// TwinCAT 3 PLC project Untitled1
// ProgramVersion: 3.1.4023.0
// libraries:
//   CmpBitmapPool, * (System)
//   Tc2_MC2, * (Beckhoff Automation GmbH)
//   Tc2_Standard, * (Beckhoff Automation GmbH)
//   Tc2_System, * (Beckhoff Automation GmbH)
//   Tc2_Utilities, * (Beckhoff Automation GmbH)
//   Tc3_Module, * (Beckhoff Automation GmbH)
// project tree:
//   DUTs/ A21ToolStorage.TcDUT (not stored), Bundle.TcDUT (not stored), EOAT.TcDUT (not stored), Interval.TcDUT (not stored), PositionMaterials.TcDUT (not stored)
//   DUTs/Enums/ A21.TcDUT (not stored), Chipboard.TcDUT (not stored), Homing.TcDUT, SectionEnum.TcDUT (not stored), Surface.TcDUT (not stored), WoodBunk.TcDUT (not stored)
//   DUTs/Insertion/Drives/ AirPiston.TcPOU (not stored), ClearLinkMC.TcPOU, SimplePiston.TcPOU (not stored)
//   DUTs/Insertion/ Insertion.TcPOU (not stored), SuctionPad.TcDUT (not stored)
//   DUTs/Insertion/Prototypes/ FBA_Drive.TcPOU (not stored), I_ContinuousDrive.TcIO (not stored), I_Drive.TcIO (not stored), I_PositionalDrive.TcIO (not stored), I_EncodedDrive.TcIO (not stored)
//   DUTs/Machines/ Conveyor.TcPOU (not stored), ConveyorMode.TcDUT (not stored), KukaRobot.TcPOU (not stored), RobotA21.TcPOU (not stored), StrapMachine.TcPOU
//   DUTs/Material Holders/ MaterialHolder.TcPOU, MaterialSlot.TcDUT, SkidMagazine.TcPOU, StagingTable.TcPOU
//   GVLs/ ContainerArrays.TcGVL, GVL.TcGVL (not stored), Hardware.TcGVL (not stored), Misc.TcGVL (not stored)
//   / PlcTask.TcTTO (not stored)
//   POUs/A21a - Chipboard/AOIs/ AOI_LoadChipboard.TcPOU
//   POUs/A21b - Wood Bunk/AOIs/ AOI_LoadWoodBunk.TcPOU, AOI_StageWoodBunk.TcPOU, AOI_StagingTemplate.TcPOU
//   POUs/ FB_System.TcPOU (not stored), MAIN.TcPOU
//   POUs/Hardware Calls/ InsertionQuality.TcPOU (not stored), SuctionQuality.TcPOU (not stored), CallHardware.TcPOU, SetSuctions.TcPOU (not stored), SetupHardware.TcPOU
//   POUs/A21a - Chipboard/ ChipboardEx.TcPOU
//   POUs/A21b - Wood Bunk/ WoodBunkEx.TcPOU
//   POUs/Utility/ AddToStringArray.TcPOU (not stored), ArrayIsEmpty.TcPOU (not stored), BoolVLArrayToInteger.TcPOU (not stored), BoolPtrArrayToInteger.TcPOU (not stored), CleanStringsArray.TcPOU (not stored), IntegerBitAccess.TcPOU (not stored), IntegerToBoolArray.TcPOU (not stored), JoinStrings.TcPOU (not stored), WithinTolerance.TcPOU (not stored)
// real-time tasks:
//   TASK PlcTask: cycle T#10ms, priority 20, ADS port 350
// I/O:
//   DEVICE Device 1 (EtherCAT) (disabled), AmsNetId 192.168.101.188.2.1
//     EK1200 [EK1200-5000 EtherCAT Power supply (2A E-Bus)]
//       IPC_O [EL2809 16Ch. Dig. Output 24V, 0.5A]
//       JUNC_A21 [EK1122 2 port EtherCAT junction]
//         C4 [EK1100 EtherCAT Coupler (2A E-Bus)]
//           C4_I1 [EL1809 16Ch. Dig. Input 24V, 3ms]
//           C4_O2 [EL2809 16Ch. Dig. Output 24V, 0.5A]
//           C4_O3 [EL2809 16Ch. Dig. Output 24V, 0.5A]
//           BRIDGE_ROBOT1 [EL6695 EtherCAT Bridge terminal (Primary)]
//           Term 14 (EL9011) [EL9011 End Terminal]
//         SB01 [EP1809-0021 16 Ch. Dig. Input 24V, 3ms, M8]
//         SB05 [EP1008-0001 8 Ch. Dig. Input 24V, 3ms, M8]
//         SB04 [EP1809-0021 16 Ch. Dig. Input 24V, 3ms, M8]
//         SB03 [EP1008-0001 8 Ch. Dig. Input 24V, 3ms, M8]
//         C1 [EK1100 EtherCAT Coupler (2A E-Bus)]
//           C1_I1 [EL1809 16Ch. Dig. Input 24V, 3ms]
//           C1_O2 [EL2809 16Ch. Dig. Output 24V, 0.5A]
//           BRIDGE_ROBOT2 [EL6695 EtherCAT Bridge terminal (Primary)]
//           Term 13 (EL9011) [EL9011 End Terminal]
//         SB02 [EP1809-0021 16 Ch. Dig. Input 24V, 3ms, M8]
//         SB07 [EP1008-0001 8 Ch. Dig. Input 24V, 3ms, M8]
//         SB06 [EP1008-0001 8 Ch. Dig. Input 24V, 3ms, M8]
// variable links:
//   Untitled1/Untitled1 Instance <-> Device 1 (EtherCAT)/EK1200/JUNC_A21/C1/BRIDGE_ROBOT2
//     PlcTask Inputs/Hardware.robot2.inputs[{2..20}] <-> IO Inputs/In_{2..20}  (19 links)
//     PlcTask Inputs/Hardware.robot2.inputs[1] <-> IO Inputs/In
//     PlcTask Inputs/Hardware.robot2.offline <-> SYNC Inputs/External device not connected
//     PlcTask Outputs/Hardware.robot2.outputs[{2..50}] <-> IO Outputs/Out_{2..50}  (49 links)
//     PlcTask Outputs/Hardware.robot2.outputs[1] <-> IO Outputs/Out
//   Untitled1/Untitled1 Instance <-> Device 1 (EtherCAT)/EK1200/JUNC_A21/C1/C1_I1
//     PlcTask Inputs/Hardware.strapperA21.atBundleLevel <-> Channel 6/Input
//     PlcTask Inputs/Hardware.strapperA21.done <-> Channel 4/Input
//     PlcTask Inputs/Hardware.strapperA21.error <-> Channel 1/Input
//     PlcTask Inputs/Hardware.strapperA21.home <-> Channel 5/Input
//     PlcTask Inputs/Hardware.strapperA21.ready <-> Channel 2/Input
//   Untitled1/Untitled1 Instance <-> Device 1 (EtherCAT)/EK1200/JUNC_A21/C1/C1_O2
//     PlcTask Outputs/Hardware.strapperA21.enable <-> Channel 2/Output
//     PlcTask Outputs/Hardware.strapperA21.execute <-> Channel 1/Output
//     PlcTask Outputs/Hardware.strapperA21.reset <-> Channel 3/Output
//   Untitled1/Untitled1 Instance <-> Device 1 (EtherCAT)/EK1200/JUNC_A21/C4/BRIDGE_ROBOT1
//     PlcTask Inputs/Hardware.robot1.inputs[{2..20}] <-> IO Inputs/In_{2..20}  (19 links)
//     PlcTask Inputs/Hardware.robot1.inputs[1] <-> IO Inputs/In
//     PlcTask Inputs/Hardware.robot1.offline <-> SYNC Inputs/External device not connected
//     PlcTask Outputs/Hardware.robot1.outputs[{2..50}] <-> IO Outputs/Out_{2..50}  (49 links)
//     PlcTask Outputs/Hardware.robot1.outputs[1] <-> IO Outputs/Out
//   Untitled1/Untitled1 Instance <-> Device 1 (EtherCAT)/EK1200/JUNC_A21/C4/C4_I1
//     PlcTask Inputs/Hardware.suctionA21Top[1].occupied <-> Channel 9/Input
//     PlcTask Inputs/Hardware.suctionA21Top[2].occupied <-> Channel 10/Input
//     PlcTask Inputs/Hardware.suctionA21Top[3].occupied <-> Channel 11/Input
//     PlcTask Inputs/Hardware.verticalDriveA21Left.home <-> Channel 3/Input
//     PlcTask Inputs/Hardware.verticalDriveA21Left.innerLimit <-> Channel 2/Input
//     PlcTask Inputs/Hardware.verticalDriveA21Left.outerLimit <-> Channel 1/Input
//     PlcTask Inputs/Hardware.verticalDriveA21Right.home <-> Channel 7/Input
//     PlcTask Inputs/Hardware.verticalDriveA21Right.innerLimit <-> Channel 6/Input
//     PlcTask Inputs/Hardware.verticalDriveA21Right.outerLimit <-> Channel 5/Input
//   Untitled1/Untitled1 Instance <-> Device 1 (EtherCAT)/EK1200/JUNC_A21/C4/C4_O2
//     PlcTask Outputs/Hardware.horizontalDriveA21Left.valveExtend <-> Channel 5/Output
//     PlcTask Outputs/Hardware.horizontalDriveA21Left.valveRetract <-> Channel 6/Output
//     PlcTask Outputs/Hardware.horizontalDriveA21Right.valveExtend <-> Channel 15/Output
//     PlcTask Outputs/Hardware.horizontalDriveA21Right.valveRetract <-> Channel 16/Output
//     PlcTask Outputs/Hardware.suctionA21Left[{1..4}].enable <-> Channel {7..10}/Output  (4 links)
//     PlcTask Outputs/Hardware.verticalDriveA21Left.brakeRelease <-> Channel 4/Output
//     PlcTask Outputs/Hardware.verticalDriveA21Right.brakeRelease <-> Channel 14/Output
//   Untitled1/Untitled1 Instance <-> Device 1 (EtherCAT)/EK1200/JUNC_A21/C4/C4_O3
//     PlcTask Outputs/Hardware.pistonA21Bottom.pistonExtend <-> Channel 5/Output
//     PlcTask Outputs/Hardware.pistonA21Bottom.pistonRetract <-> Channel 6/Output
//     PlcTask Outputs/Hardware.suctionA21Bottom[1].enable <-> Channel 7/Output
//     PlcTask Outputs/Hardware.suctionA21Bottom[2].enable <-> Channel 8/Output
//     PlcTask Outputs/Hardware.suctionA21Right[{1..4}].enable <-> Channel {1..4}/Output  (4 links)
//     PlcTask Outputs/Hardware.suctionA21Top[1].enable <-> Channel 9/Output
//     PlcTask Outputs/Hardware.suctionA21Top[2].enable <-> Channel 10/Output
//     PlcTask Outputs/Hardware.suctionA21Top[3].enable <-> Channel 11/Output
//   Untitled1/Untitled1 Instance <-> Device 1 (EtherCAT)/EK1200/JUNC_A21/SB01
//     PlcTask Inputs/ContainerArrays.tableOccupancyA21Left[{1..10}] <-> Channel {1..10}/Input  (10 links)
//     PlcTask Inputs/Hardware.horizontalDriveA21Left.home <-> Channel 11/Input
//     PlcTask Inputs/Hardware.horizontalDriveA21Left.innerLimit <-> Channel 12/Input
//     PlcTask Inputs/Hardware.suctionA21Left[{1..4}].occupied <-> Channel {13..16}/Input  (4 links)
//   Untitled1/Untitled1 Instance <-> Device 1 (EtherCAT)/EK1200/JUNC_A21/SB02
//     PlcTask Inputs/ContainerArrays.tableOccupancyA21Right[{1..10}] <-> Channel {1..10}/Input  (10 links)
//     PlcTask Inputs/Hardware.horizontalDriveA21Right.home <-> Channel 11/Input
//     PlcTask Inputs/Hardware.horizontalDriveA21Right.innerLimit <-> Channel 12/Input
//     PlcTask Inputs/Hardware.suctionA21Right[{1..4}].occupied <-> Channel {13..16}/Input  (4 links)
//   Untitled1/Untitled1 Instance <-> Device 1 (EtherCAT)/EK1200/JUNC_A21/SB07
//     PlcTask Inputs/Hardware.pistonA21Bottom.extended <-> Channel 5/Input
//     PlcTask Inputs/Hardware.pistonA21Bottom.retracted <-> Channel 4/Input
//     PlcTask Inputs/Hardware.suctionA21Bottom[1].occupied <-> Channel 6/Input
//     PlcTask Inputs/Hardware.suctionA21Bottom[2].occupied <-> Channel 7/Input

// ---- DUTs/Enums/Homing.TcDUT
{attribute 'qualified_only'}
{attribute 'strict'}
TYPE Homing :
(
	IDLE,
	IN,
	OUT,
	OUT_FINAL,
	STOP,
	SET,
	DONE,
	
	size
);
END_TYPE

// ---- DUTs/Material Holders/MaterialSlot.TcDUT
TYPE MaterialSlot :
STRUCT
	material : REFERENCE TO STRING;
	occupied : REFERENCE TO BOOL;
END_STRUCT
END_TYPE

// ---- GVLs/ContainerArrays.TcGVL
//{attribute 'qualified_only'}
VAR_GLOBAL //data arrays to be passed into material holder FBs - direct access is strongly discouraged
	
	skidSlotsA21Left, skidSlotsA21Right : ARRAY[1..2] OF STRING; //chipboard skid
	skidOccupancyA21Left, skidOccupancyA21Right : ARRAY[1..2] OF BOOL;
	
	magazineSlotsA21Left, magazineSlotsA21Right : ARRAY[1..15] OF STRING; //wood bunk magazine
	magazineOccupancyA21Left, magazineOccupancyA21Right : ARRAY[1..15] OF BOOL;
	
	tableSlotsA21Left, tableSlotsA21Right : ARRAY[1..10] OF STRING; //staging table
	tableOccupancyA21Left, tableOccupancyA21Right AT %I* : ARRAY[1..10] OF BOOL;
	
	skidHmiA21Left, skidHmiA21Right AT %M* : ARRAY[1..2] OF MaterialSlot;
	magazineHmiA21Left, magazineHmiA21Right AT %M* : ARRAY[1..15] OF MaterialSlot;
	tableHmiA21Left : ARRAY[1..10] OF MaterialSlot; (*:= [
		(material := 'WDS20', occupied := TRUE), 
		(material := 'WDS20', occupied := TRUE), 
		(material := 'WDS20', occupied := TRUE), 
		(material := 'WDS20', occupied := TRUE)];*)
	tableHmiA21Right : ARRAY[1..10] OF MaterialSlot; (*:= [
		(material := 'WDS20', occupied := TRUE), 
		(material := 'WDB20', occupied := TRUE), 
		(material := 'WDS20', occupied := TRUE), 
		(material := 'WDB20', occupied := TRUE)];*)
	
END_VAR

// ---- DUTs/Insertion/Drives/ClearLinkMC.TcPOU
FUNCTION_BLOCK ClearLinkMC EXTENDS FBA_Drive IMPLEMENTS I_EncodedDrive //I_PositionalDrive, I_ContinuousDrive
VAR_OUTPUT
	pulse AT %Q* : INT; //num pulses
	outputRegister AT %Q* : INT;
	brakeRelease AT %Q* : BOOL;
	
	A : BOOL; //direction (F = inwards, T = outwards)
	B : BOOL; //home bit
	clear : BOOL;
	
	hlfb AT %I* : REAL; //high level feedback, if -9999 then servo is idle
	position, targetPos : LREAL;
END_VAR
VAR
	pulseRequest : INT;
	
	minHoming : TON;
	resetTimer : TP;
	
	mode : (DISABLE, HOLD, TARGET, CONTINUOUS, RESET_ERR);
END_VAR
VAR_STAT CONSTANT
	resetTime : TIME := T#1000MS;
	unitsPerPulse : INT := 800; //800 Teknic units per revolution
	distancePerPulse : INT := 5; //5mm per revolution
END_VAR

//M-connector output register
outputRegister.0 := bEnable; 	//enable
outputRegister.1 := A; 			//direction bit
outputRegister.2 := B; 			//homing bit - set to TRUE after startup to begin homing, then set to FALSE to finish homing
outputRegister.3 := clear; 		//reset bit

resetTimer(IN:= , PT:= resetTime, Q=> clear, ET=> ); //reset timer

IF NOT bEnable THEN
	homingComplete := FALSE;
	mode := HOLD;
END_IF

override(); //if sensor limits are reached, this method blocks motion that would exceed the limits

CASE mode OF		
	HOLD: //hold current position, no motion
		pulse := 0;
		pulseRequest := 0;
	
	TARGET:	//target a given position
		IF WithinTolerance(position, targetPos, distancePerPulse) THEN
			pulseRequest := 0;
			mode := HOLD;
			
		ELSIF NOT Busy THEN
			A :=  position < targetPos;
			//pulseRequest := TO_INT(ABS(position - targetPos)/distancePerPulse);
			pulseRequest := 1;
			
		END_IF
		
	CONTINUOUS: //single pulses in the direction specified by moveContinuous()
		pulseRequest := 1;
		
	RESET_ERR: //reset pulse, servo may need to be rehomed aftewards
		pulse := 0;
		pulseRequest := 0;
		resetTimer.IN := TRUE;
		
		IF resetTimer.Q THEN
			resetTimer.IN := FALSE;
			mode := HOLD;
		END_IF
		
END_CASE

sequence();

PROPERTY Busy : BOOL
GET
Busy := hlfb <> -9999;
END_GET
END_PROPERTY

PROPERTY CurrentPosition : LREAL
GET
CurrentPosition := position;
END_GET
SET
position := CurrentPosition;
END_SET
END_PROPERTY

PROPERTY Error : BOOL
GET
END_GET
END_PROPERTY

METHOD homingSequence : BOOL
minHoming(IN:= , PT:= T#1S, Q=> , ET=> ); //IN and OUT should be held for at least 1 second - may be removed for deployment

IF NOT bEnable THEN //homing does not begin until software enable
	RETURN;
END_IF

CASE step OF
	Homing.IDLE:
		bEnable := FALSE;
		A := FALSE;
		B := FALSE;
		brakeRelease := TRUE;
		
		homingComplete := FALSE;
		step := Homing.IN;
		
	Homing.IN: //let insertion drop to inner limit before homing
		bEnable := FALSE;
		A := FALSE;
		B := FALSE;
		brakeRelease := TRUE;
		
		minHoming.IN := TRUE;
		
		IF NOT innerLimit AND minHoming.Q THEN
			minHoming.IN := FALSE;
			step := Homing.OUT;
		END_IF
	
	Homing.OUT:
		bEnable := TRUE;
		A := FALSE;
		B := TRUE;
		brakeRelease := TRUE;
		
		minHoming.IN := TRUE;
		
		IF NOT home AND minHoming.Q THEN
			minHoming.IN := FALSE;
			step := Homing.DONE;
		END_IF
		
	Homing.DONE:
		bEnable := TRUE;
		A := FALSE;
		B := FALSE;
		brakeRelease := TRUE;
			
		position := 0;
		
		homingComplete := TRUE;
		homingSequence := TRUE;
		
		mode := HOLD;
		step := Homing.IDLE;
	
END_CASE
END_METHOD

METHOD moveAbsolute : BOOL
VAR_INPUT
	newTarget : LREAL;
END_VAR
targetPos := newTarget;
mode := TARGET;
END_METHOD

METHOD moveContinuous : BOOL
VAR_INPUT
	direction : MC_Direction;
END_VAR
IF direction = MC_Negative_Direction THEN
	A := FALSE;
ELSIF direction = MC_Positive_Direction THEN
	A := TRUE;
END_IF

mode := CONTINUOUS;
END_METHOD

METHOD moveRelative : BOOL
VAR_INPUT
	distance : LREAL;
END_VAR
targetPos := targetPos + distance;

mode := TARGET;
END_METHOD

METHOD PRIVATE override : BOOL
VAR_INPUT
END_VAR
(*
IF (*NOT*) home THEN //block outwards motion
	position := 0;
	IF A THEN
		mode := HOLD;
	END_IF
	
ELSIF (*NOT*) outerLimit AND_THEN A THEN //block outwards motion
	mode := HOLD;

ELSIF (*NOT*) innerLimit AND_THEN NOT A THEN //block inwards motion
	mode := HOLD;
	
END_IF
*)


IF
	((*NOT*) home AND_THEN A) OR
	((*NOT*) outerLimit AND_THEN A) OR
	((*NOT*) innerLimit AND_THEN NOT A)
THEN
	mode := HOLD;
END_IF


IF (*NOT*) home THEN //block outwards motion
	position := 0;
END_IF
END_METHOD

METHOD reset : BOOL
VAR_INPUT
END_VAR
mode := RESET_ERR;
END_METHOD

METHOD PRIVATE sequence : BOOL
VAR_INPUT
END_VAR
IF Busy THEN //servo is active
	IF A THEN //positive direction
		position := position + (distancePerPulse * pulse);
	ELSE //negative direction
		position := position - (distancePerPulse * pulse);
	END_IF
	pulse := 0; //pulses already received, can be set to 0 so position change is not compounded

ELSIF pulse = 0 THEN //servo is not active
	pulse := pulseRequest;
	pulseRequest := 0; //remove this if not working as intended
	
END_IF
END_METHOD

METHOD stop : BOOL
VAR_INPUT
END_VAR
mode := HOLD;
END_METHOD

PROPERTY TargetPosition : LREAL
GET
END_GET
SET
targetPos := TargetPosition;
END_SET
END_PROPERTY

END_FUNCTION_BLOCK

// ---- DUTs/Machines/StrapMachine.TcPOU
FUNCTION_BLOCK StrapMachine
VAR_INPUT
	bEnable : BOOL;
END_VAR
VAR_OUTPUT
	enable AT %Q* : BOOL;
	execute AT %Q* : BOOL;
	reset AT %Q* : BOOL;
	
	error AT %I* : BOOL;
	ready AT %I* : BOOL;
	//busy (*AT %I**) : BOOL;
	done AT %I* : BOOL;
	home AT %I* : BOOL;
	
	timeout : BOOL;
	
	atBundleLevel AT %I* : BOOL;
END_VAR
VAR	
	holdPost : TON;
	delay : TON;
	
	start : BOOL;
	step : (SETUP, RUN, WAIT);
END_VAR
VAR_STAT CONSTANT
	pulseTime : TIME := T#100MS;
	holdTime : TIME := T#500MS;
	maxDelay : TIME := T#30S;
END_VAR

holdPost(IN:= , PT:= holdTime, Q=> , ET=> );
delay(IN:= step > 0 OR start, PT:= maxDelay, Q=> timeout, ET=> );

IF delay.Q THEN
	delay.IN := FALSE;
	//timeout := TRUE;
	//busy := FALSE;
	
	start := FALSE;
	step := SETUP;
END_IF

enable := bEnable AND robot1.strapSafetyIn AND robot2.strapSafetyIn;

CASE step OF
	SETUP:
		//busy := FALSE;
		IF error THEN
			enable := FALSE;
			execute := FALSE;
			clear();
			
		ELSIF start AND enable THEN //strapping does not start if error
			start := FALSE;
			step := RUN;
		END_IF
	
	RUN:
		IF NOT execute THEN
			execute := TRUE;
			RETURN; //keeps execute TRUE for at least 1 cycle
		END_IF
		
		IF execute AND NOT ready (*AND NOT home*) THEN
			execute := FALSE;
			step := WAIT;
		END_IF
		
	WAIT: //due to the use of DC motors instead of stepper motors in the machine, a short delay is required before next strap
		IF home THEN
			holdPost.IN := TRUE;
			enable := FALSE;
			execute := FALSE;
		END_IF
		
		IF holdPost.Q THEN
			holdPost.IN := FALSE;
			done := TRUE;
			step := 0;
		END_IF
		
END_CASE

(*
executePulse(IN:= , PT:= pulseTime, Q=> , ET=> );
execute := executePulse.IN AND NOT executePulse.Q;

IF executePulse.Q THEN
	executePulse.IN := FALSE;
END_IF


resetPulse(IN:= , PT:= pulseTime, Q=> , ET=> );
StrapMachineST.reset := resetPulse.IN AND NOT resetPulse.Q;

IF resetPulse.Q THEN
	executePulse.IN := FALSE;
END_IF

ready := enable AND NOT execute AND NOT StrapMachineST.reset AND NOT error AND home;
*)

METHOD clear : BOOL
VAR_INPUT
END_VAR
(*
reset should be continuously called until machine returns evidence that it is ready again
machine is expected to not respond to reset signals if it is already in an idle state
*)
enable := FALSE;
execute := FALSE;

IF error THEN
	reset := NOT reset;
ELSE
	reset := FALSE;
END_IF

clear := NOT error;
END_METHOD

METHOD strap : BOOL
VAR_INPUT
END_VAR
//IF ready AND NOT busy AND NOT error THEN
	//busy := TRUE;
	//start := TRUE;
	//strap := TRUE;
//END_IF

start := TRUE;
END_METHOD

END_FUNCTION_BLOCK

// ---- DUTs/Material Holders/MaterialHolder.TcPOU
FUNCTION_BLOCK MaterialHolder
VAR_IN_OUT
	slots : ARRAY[*] OF STRING;
	occupied : ARRAY[*] OF BOOL;
	
	hmiTable : ARRAY[*] OF MaterialSlot;
END_VAR
VAR
	numSlots : INT;
END_VAR

(*
by default:
	hmiTable contains the slot names, occupied[] contains the occupancy data
	slots[] cyclically copies data from hmiTable
	hmiTable cyclically copies data from occupied[]

if hmiTable is NULL (not passed in), then slots and occupied will store the true data
	
the program will access data using slots/occupied via methods
when the data is changed, data is copied from slots/occupied to hmiTable

this ensures that the methods update the HMI, and the HMI updates the data
*)


IF hmiTable <> 0 AND_THEN (slots <> 0  AND occupied <> 0) THEN
	refreshHmiTable();
END_IF

numSlots := TO_INT(UPPER_BOUND(slots, 1) - LOWER_BOUND(slots, 1) + 1);

METHOD clear : BOOL
VAR_INPUT
END_VAR
MEMSET(ADR(slots), 0, SIZEOF(slots));

IF hmiTable <> 0 THEN
	writeHmiTable();
END_IF
END_METHOD

METHOD findSlot : BOOL
VAR_INPUT
	materialID : STRING;
END_VAR
VAR_OUTPUT
	index : INT := -1;
END_VAR
VAR
	i : DINT;
END_VAR
(*
IF materialID = '' THEN
	RETURN;
END_IF
*)
FOR i:=LOWER_BOUND(slots, 1) TO UPPER_BOUND(slots, 1) BY 1 DO
	IF slots[i] = materialID THEN
		index := TO_INT(i);
		findSlot := TRUE;
		RETURN;
	END_IF
END_FOR
END_METHOD

METHOD getSlot : STRING
VAR_INPUT
	i : DINT;
END_VAR
VAR_OUTPUT
	error : BOOL;
END_VAR
error := i < LOWER_BOUND(slots, 1) OR i > UPPER_BOUND(slots, 1) (*OR slots = 0*);

IF error THEN
	RETURN;
END_IF

getSlot := slots[i];
END_METHOD

METHOD getSlotsAsArray : POINTER TO STRING
getSlotsAsArray := ADR(slots);
END_METHOD

METHOD isOccupied : BOOL
VAR_INPUT
	i : DINT;
END_VAR
VAR_OUTPUT
	errorBounds : BOOL;
END_VAR
errorBounds := i < LOWER_BOUND(slots, 1) OR i > UPPER_BOUND(slots, 1);

IF errorBounds THEN
	RETURN;
END_IF

isOccupied := occupied[i];
END_METHOD

METHOD PROTECTED refreshHmiTable : BOOL
VAR
	i : DINT;
END_VAR
FOR i:=LOWER_BOUND(hmiTable, 1) TO UPPER_BOUND(hmiTable, 1) BY 1 DO
	slots[i] := hmiTable[i].material; //slots[] copies from hmiTable
	hmiTable[i].occupied := occupied[i]; //hmiTable copies from occupied[]
END_FOR
END_METHOD

METHOD setSlots : BOOL
VAR_IN_OUT
	newSlots : ARRAY[*] OF STRING;
END_VAR
VAR
	i : DINT;
	j : DINT;
END_VAR
{warning disable C0195}
MEMCPY(
	slots, 
	newSlots, 
	SIZEOF(STRING) * MIN(
		(1 + UPPER_BOUND(newSlots, 1) - LOWER_BOUND(newSlots, 1)),
		(1 + UPPER_BOUND(slots, 1) - LOWER_BOUND(slots, 1))
	));
	
IF hmiTable <> 0 THEN
	writeHmiTable();
END_IF
END_METHOD

METHOD PROTECTED writeArrays : BOOL
VAR
	i : DINT;
END_VAR
FOR i:=LOWER_BOUND(hmiTable, 1) TO UPPER_BOUND(hmiTable, 1) BY 1 DO
	slots[i] := hmiTable[i].material;
	//occupied[i] := hmiTable[i].occupied;
END_FOR
END_METHOD

METHOD PROTECTED writeHmiTable : BOOL
VAR
	i : DINT;
END_VAR
FOR i:=LOWER_BOUND(hmiTable, 1) TO UPPER_BOUND(hmiTable, 1) BY 1 DO
	hmiTable[i].material := slots[i];
	hmiTable[i].occupied := occupied[i];
END_FOR
END_METHOD

END_FUNCTION_BLOCK

// ---- DUTs/Material Holders/SkidMagazine.TcPOU
FUNCTION_BLOCK SkidMagazine EXTENDS MaterialHolder
VAR_OUTPUT
	inPosition AT %I* : ARRAY[1..2] OF BOOL;
END_VAR

SUPER^();

METHOD setOccupancy : BOOL
VAR_INPUT
	i : INT;
	occupancy : BOOL;
END_VAR
VAR_OUTPUT
	errorBounds : BOOL;
END_VAR
errorBounds := i < LOWER_BOUND(slots, 1) OR i > UPPER_BOUND(slots, 1);

IF NOT errorBounds THEN
	occupied[i] := occupancy;
END_IF

IF hmiTable <> 0 THEN
	writeHmiTable();
END_IF
END_METHOD

END_FUNCTION_BLOCK

// ---- DUTs/Material Holders/StagingTable.TcPOU
FUNCTION_BLOCK StagingTable EXTENDS MaterialHolder

SUPER^();

METHOD autofill : BOOL
VAR_INPUT
	materialID : STRING;
END_VAR
VAR
	i : INT;
	slot : INT;
END_VAR
(*
this method will automatically find an open slot
*)
IF isFull() OR materialID = '' THEN
	RETURN;
END_IF

IF findOpenSlot(materialID, openSlot=> slot) THEN
	place(slot, materialID);
	autofill := TRUE;
END_IF

IF hmiTable <> 0 THEN
	writeHmiTable();
END_IF
END_METHOD

METHOD findOpenSlot : BOOL
VAR_INPUT
	materialID : STRING;
END_VAR
VAR_OUTPUT
	openSlot : INT := 0;
END_VAR
VAR
	i : INT;
END_VAR
IF FIND(materialID, 'WDW') > 0 THEN //top wide, load in slot 9-10
	FOR i:=9 TO 10 BY 1 DO
		IF slots[i] = '' THEN
			findOpenSlot := TRUE;
			openSlot := i;
			RETURN;
		END_IF
	END_FOR
	
//ELSIF FIND(materialID, 'WDT') > 0 OR FIND(materialID, 'WDS') > 0 THEN //standard width, load in slot 3-10
ELSIF FIND(materialID, 'WD') > 0 THEN //standard width, load in slot 1-8
	FOR i:=1 TO 8 BY 1 DO
		IF slots[i] = '' THEN
			findOpenSlot := TRUE;
			openSlot := i;
			RETURN;
		END_IF
	END_FOR
	
END_IF
END_METHOD

METHOD isEmpty : BOOL
VAR
	i : INT;
	temp : BOOL;
END_VAR
FOR i:=1 TO numSlots BY 1 DO
	temp := temp OR occupied[i]; //TRUE if any slots are occupied
END_FOR

isEmpty := NOT temp; //invert result - FALSE if any slots are occupied
END_METHOD

METHOD isFull : BOOL
VAR
	i : INT;
	temp : BOOL := TRUE;
END_VAR
FOR i:=1 TO numSlots BY 1 DO
	temp := temp AND occupied[i];
END_FOR

isFull := temp;
END_METHOD

METHOD place : BOOL
VAR_INPUT
	i : INT;
	materialID : STRING;
END_VAR
IF slots[i] = '' THEN
	slots[i] := materialID;
	place := TRUE;
END_IF

IF hmiTable <> 0 THEN
	writeHmiTable();
END_IF
END_METHOD

METHOD remove : BOOL
VAR_INPUT
	i : INT;
END_VAR
VAR_OUTPUT
	materialID : STRING;
END_VAR
remove := slots[i] <> '';

materialID := slots[i];
slots[i] := '';

IF hmiTable <> 0 THEN
	writeHmiTable();
END_IF
END_METHOD

END_FUNCTION_BLOCK

// ---- POUs/A21a - Chipboard/AOIs/AOI_LoadChipboard.TcPOU
FUNCTION_BLOCK AOI_LoadChipboard
VAR_IN_OUT CONSTANT
	sectionID : SectionEnum;
END_VAR
VAR_INPUT
	execute : BOOL;
END_VAR
VAR_IN_OUT
	robot : RobotA21;
	storage : SkidMagazine;
	loadedMaterials : ARRAY[*] OF STRING;
END_VAR
VAR_INPUT
	surfaceID : Surface;
	material : STRING;
END_VAR
VAR_OUTPUT
	busy : BOOL;
	done : BOOL;
	error : BOOL;
	
	recoveryMode : BOOL;
	failCounter : INT;
END_VAR
VAR
	run : BOOL;
	trigger : R_TRIG;
	
	step : (IDLE, PREP_ROBOT, RETRACT_CONVEYORS, GET_FROM_SKID, LOAD_TO_BUNDLE, COMPLETE);
	column : INT;
END_VAR
VAR CONSTANT
	suctionDistance : INT := 10;
END_VAR

{warning disable C0371}
IF material = '' THEN
	done := TRUE;
	RETURN;
END_IF

IF robot.error THEN
	error := TRUE;
	RETURN;
ELSIF robot.reservation <> sectionID (*AND_THEN NOT robot.reserve(sectionID)*) THEN
	RETURN;
ELSIF robot.tool <> sectionID (*AND_THEN NOT robot.changeEOAT(targetTool := sectionID)*) THEN
	RETURN;
END_IF

trigger(CLK:= execute, Q=> run);

CASE step OF
	IDLE:
		recoveryMode := FALSE;
		IF run THEN
			done := FALSE;
			error := FALSE;
			step := PREP_ROBOT;
		END_IF
	
	PREP_ROBOT:
		robot.clearCommand();
		IF robot.Ready THEN
			step := RETRACT_CONVEYORS;
		END_IF
	
	RETRACT_CONVEYORS:
		IF surfaceID = Surface.BOTTOM (*AND_THEN conveyors not retracted*) THEN
			//retract conveyors
			RETURN;
		END_IF
		step := GET_FROM_SKID;
		
	GET_FROM_SKID: //grab from chipboard skid
		IF NOT storage.findSlot(materialID := material, index => column) THEN
			error := TRUE;
			RETURN;
		(*
		ELSIF surfaceID = Surface.BOTTOM (*AND_THEN (*conveyor not lowered*)*) THEN
			//lower conveyor
			RETURN;
		*)
		END_IF
		
		IF robot.eoatDistance < suctionDistance THEN
			robot.HoldMaterial := storage.getSlot(i := column);
		END_IF
		
		IF robot.Done THEN
			step := COMPLETE;
			RETURN;
		ELSIF robot.materialAtHoldingPosition.4 OR robot.materialAtHoldingPosition.5 THEN //bits 4 and 5 are chipboard in position
			step := LOAD_TO_BUNDLE;
			RETURN;
		END_IF
		
		robot.setGroup(group := 1, value := A21.PLACE_CHIPBOARD_TOP);
		robot.setGroup(group := 2, value := column);
		
	LOAD_TO_BUNDLE: //place to bundle
		IF robot.Done THEN
			step := COMPLETE;
			RETURN;
		END_IF
		
		IF robot.HoldMaterial <> '' THEN
			loadedMaterials[surfaceID] := robot.HoldMaterial;
			robot.HoldMaterial := '';
		END_IF
		
	COMPLETE:
		IF loadedMaterials[surfaceID] = material THEN
			done := TRUE;
			failCounter := 0;
		ELSE
			error := TRUE;
			failCounter := failCounter + 1;
		END_IF
		step := 0;
END_CASE

busy := run OR step > 0;

END_FUNCTION_BLOCK

// ---- POUs/A21b - Wood Bunk/AOIs/AOI_LoadWoodBunk.TcPOU
FUNCTION_BLOCK AOI_LoadWoodBunk
VAR_IN_OUT CONSTANT
	sectionID : SectionEnum;
END_VAR
VAR_INPUT
	execute : BOOL;
END_VAR
VAR_IN_OUT
	robot : RobotA21;
	table : StagingTable;
	suctions : ARRAY[*] OF SuctionPad;
	loadedMaterials : ARRAY[*] OF STRING;
END_VAR
VAR_INPUT
	surfaceID : Surface;
	material : STRING;
END_VAR
VAR_OUTPUT
	busy : BOOL;
	done : BOOL;
	error : BOOL;
	
	recovery : BOOL;
	failCounter : INT;
END_VAR
VAR
	run : BOOL;
	trigger : R_TRIG;
	
	slot : INT;
	
	suctionTimer : TON;
	step : (IDLE, PREP_ROBOT, GET_FROM_TABLE, LOAD_TO_INSERTION, COMPLETE, RECOVERY_IDLE, RECOVERY_REMOVE, RECOVERY_WAIT, RECOVERY_STAGE);
END_VAR
VAR CONSTANT
	suctionDelay : TIME := T#2S;
END_VAR

{warning disable C0371}

trigger(CLK:= execute, Q=> );
busy := trigger.Q OR step > 0;

IF step > IDLE AND_THEN NOT preExecution() THEN //conditions to track before execution
	RETURN;
END_IF

(*
if required bunk was not found on table - restage entire table
if bunk was not loaded correctly - remove bunk, then restage entire table
*)
CASE step OF
	IDLE:
		IF trigger.Q THEN
			recovery := FALSE;
			done := FALSE;
			error := FALSE;
			step := PREP_ROBOT;
		END_IF
		
	PREP_ROBOT:
		robot.clearCommand();
		IF robot.Ready THEN
			step := GET_FROM_TABLE;
			slot := 0;
		END_IF
		
	GET_FROM_TABLE:		
		IF slot < 1 AND_THEN NOT table.findSlot(materialID := material, index => slot) THEN
			step := RECOVERY_STAGE;
			RETURN;
		END_IF
		
		IF NOT table.isOccupied(i := slot) AND table.getSlot(i := slot) <> '' THEN //move from table to robot gripper
			robot.HoldMaterial := table.getSlot(i := slot);
			table.remove(i := slot, materialID => );
		END_IF
		
		IF robot.Done THEN
			step := COMPLETE;
			RETURN;
		ELSIF robot.materialAtHoldingPosition >= 1 AND robot.materialAtHoldingPosition <= 8 THEN
			step := LOAD_TO_INSERTION;
			RETURN;
		END_IF
		
		CASE surfaceID OF
			Surface.TOP: 					robot.setGroup(group := 1, value := A21.LOAD_BUNK_TOP); 
			Surface.LEFT, Surface.RIGHT: 	robot.setGroup(group := 1, value := A21.LOAD_BUNK_SIDE);
			Surface.BOTTOM: 				robot.setGroup(group := 1, value := A21.LOAD_BUNK_BOTTOM);
		END_CASE
		robot.setGroup(group := 2, value := slot); 
			
	LOAD_TO_INSERTION:
		IF robot.materialAtHoldingPosition > 0 AND robot.HoldMaterial <> '' THEN //move from gripper to insertion
			IF loadedMaterials[surfaceID] = '' THEN //transfer to insertion as is
				loadedMaterials[surfaceID] := robot.HoldMaterial;
			ELSE //join with existing material using underscore _
				loadedMaterials[surfaceID] := JoinStrings(loadedMaterials[surfaceID], robot.HoldMaterial, '_');
			END_IF
			robot.HoldMaterial := '';
		END_IF
		
		CASE surfaceID OF
			Surface.TOP, Surface.BOTTOM:	SetSuctions(suctions, TRUE);
			Surface.LEFT, Surface.RIGHT:	SetSuctions(suctions, TRUE );
		END_CASE
		
		IF robot.Done THEN
			suctionTimer.IN := FALSE;
			step := COMPLETE;
			RETURN;
		END_IF
		
		suctionTimer(IN:= , PT:= suctionDelay, Q=> , ET=> );
		suctionTimer.IN := TRUE;
		
		IF suctionTimer.Q THEN
			robot.setGroup(group := 9, value := robot.materialAtHoldingPosition);
		END_IF
	
	COMPLETE:
		robot.clearCommand();
		
		//check insertion quality
		IF InsertionQuality(suctions := suctions, insertionMaterial := loadedMaterials[surfaceID], recipeMaterial := material) THEN
			done := TRUE;
			slot := 0;
			step := 0;
		ELSE //recovery - restage table
			failCounter := failCounter + 1;
			step := RECOVERY_IDLE;
		END_IF
		
	//---------RECOVERY-----------------------------------------
	RECOVERY_IDLE:
		robot.clearCommand();
		IF robot.Ready THEN
			step := RECOVERY_REMOVE;
		END_IF
		
	RECOVERY_REMOVE:
		IF robot.Done THEN
			//step := RECOVERY_WAIT;
			step := RECOVERY_STAGE;
			RETURN;
		END_IF
		
		CASE surfaceID OF
			Surface.TOP:					robot.setGroup(group := 1, value := A21.REMOVE_BUNK_TOP);
			Surface.LEFT, Surface.RIGHT:	robot.setGroup(group := 1, value := A21.REMOVE_BUNK_SIDE);
			Surface.BOTTOM:					robot.setGroup(group := 1, value := A21.REMOVE_BUNK_BOTTOM);
		END_CASE
	
	RECOVERY_WAIT: //this step is unused for now
		robot.clearCommand();
		IF robot.Ready THEN
			step := RECOVERY_STAGE;
		END_IF
	
	RECOVERY_STAGE:	
		recovery := TRUE;
		error := TRUE;
		
END_CASE

METHOD PRIVATE preExecution : BOOL
VAR_INPUT
END_VAR
{warning disable C0371}
IF material = '' THEN
	done := TRUE;
	RETURN;
END_IF

IF //robot must be ready before execution
	robot.error OR 
	robot.reservation <> sectionID OR 
	robot.tool <> sectionID
THEN
	error := TRUE;
	RETURN;
END_IF

preExecution := TRUE;
END_METHOD

METHOD reset : BOOL
VAR_INPUT
END_VAR
VAR
	temp : AOI_LoadWoodBunk;
END_VAR
//(*
done := FALSE;
error := FALSE;
recovery := FALSE;
slot := 0;
step := 0;

failCounter := 0;
//*)
//THIS^ := temp;
END_METHOD

END_FUNCTION_BLOCK

// ---- POUs/MAIN.TcPOU
PROGRAM MAIN
VAR
	stop : BOOL;
	manualStep : BOOL := TRUE;
	manualSuction : BOOL;
	
	moduleWB : WoodBunkEx;
	moduleCIP : ChipboardEx;
	
	exec1 : BOOL;
	exec2 : BOOL;
END_VAR

CallHardware(); //start program with hardware call - pass values and arrays into function blocks
SetupHardware(); //initialize values

runModules(); //LLD

CallHardware(); //end program with hardware call

ACTION runModules:
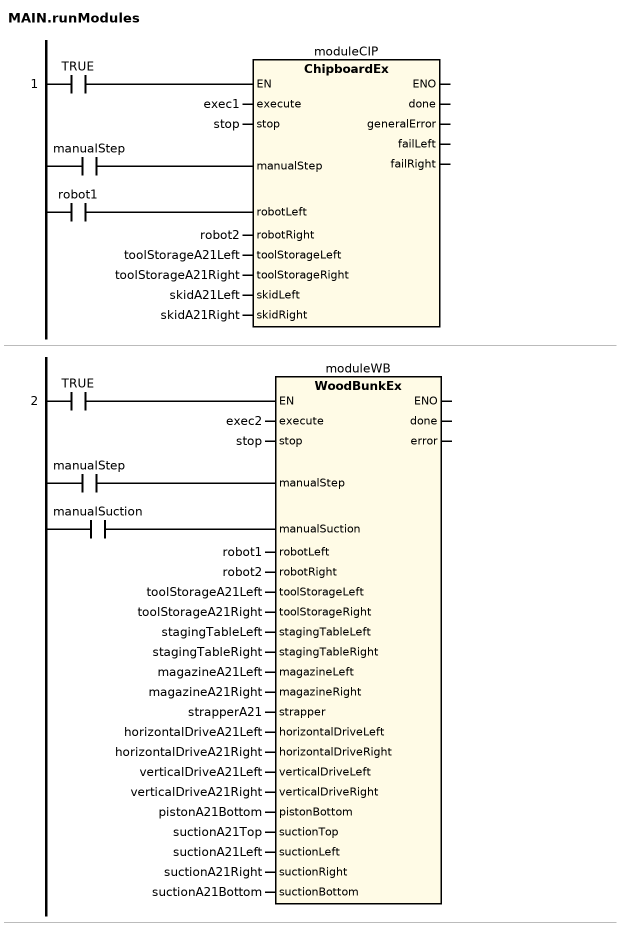
// NETWORK 1
moduleCIP(
    execute := exec1,
    stop := stop,
    manualStep := manualStep,
    robotLeft := robot1,
    robotRight := robot2,
    toolStorageLeft := toolStorageA21Left,
    toolStorageRight := toolStorageA21Right,
    skidLeft := skidA21Left,
    skidRight := skidA21Right); // ChipboardEx

// NETWORK 2
moduleWB(
    execute := exec2,
    stop := stop,
    manualStep := manualStep,
    manualSuction := manualSuction,
    robotLeft := robot1,
    robotRight := robot2,
    toolStorageLeft := toolStorageA21Left,
    toolStorageRight := toolStorageA21Right,
    stagingTableLeft := stagingTableLeft,
    stagingTableRight := stagingTableRight,
    magazineLeft := magazineA21Left,
    magazineRight := magazineA21Right,
    strapper := strapperA21,
    horizontalDriveLeft := horizontalDriveA21Left,
    horizontalDriveRight := horizontalDriveA21Right,
    verticalDriveLeft := verticalDriveA21Left,
    verticalDriveRight := verticalDriveA21Right,
    pistonBottom := pistonA21Bottom,
    suctionTop := suctionA21Top,
    suctionLeft := suctionA21Left,
    suctionRight := suctionA21Right,
    suctionBottom := suctionA21Bottom); // WoodBunkEx
END_ACTION

END_PROGRAM

// ---- POUs/A21b - Wood Bunk/WoodBunkEx.TcPOU
FUNCTION_BLOCK WoodBunkEx
VAR_IN_OUT //controls
	execute : BOOL;
	stop : BOOL;
	
	manualStep : BOOL;
	manualSuction : BOOL;
END_VAR
VAR_IN_OUT //references to required hardware
	robotLeft, robotRight : RobotA21;
	toolStorageLeft, toolStorageRight : A21ToolStorage;
	
	stagingTableLeft, stagingTableRight : StagingTable;
	magazineLeft, magazineRight : SkidMagazine;
	
	strapper : StrapMachine;
	
	horizontalDriveLeft, horizontalDriveRight : AirPiston;
	verticalDriveLeft, verticalDriveRight : ClearLinkMC;
	pistonBottom : SimplePiston;
	
	suctionTop : ARRAY[*] OF SuctionPad; (*1..3*)
	suctionLeft : ARRAY[*] OF SuctionPad; (*1..4*)
	suctionRight : ARRAY[*] OF SuctionPad; (*1..4*)
	suctionBottom : ARRAY[*] OF SuctionPad; (*1..2*)
END_VAR
VAR_OUTPUT
	//ready : BOOL;
	done : BOOL;
	error : BOOL;
END_VAR
VAR //for testing, to be removed when deployoed
	latchLeft, latchRight : BOOL; //prevents SMC sliders from overshooting
	suctionEnableTop, suctionEnableLeft, suctionEnableRight, suctionEnableBottom : BOOL;
END_VAR
VAR //Allen-Bradley-style AOIs encapsulate functionality and reduce the number of module variables	
	step : (IDLE, STAGING, LOAD_WB, PUSH, STRAP, RELEASE, COMPLETE := 1050);
	iPair : INT;
	
	loadStep : INT;
	stageStep : INT;
	
	stageStepLeft, stageStepRight : INT;
	//iSlotLeft, iSlotRight : INT;
END_VAR
VAR //local types
	demoHeight : REAL := 600; //mm
	materialsArr : ARRAY[0..GVL.maxPairs] OF PositionMaterials := [
		( position := 0, top := 'WDS20', left := 'WDS20', right := 'WDS20', bottom := 'WDB20' ),
		( position := 69, top := 'WDS20', left := 'WDS20', right := 'WDS20', bottom := 'WDB20' )
	];
	
	insertionLeft, insertionRight : Insertion;
	loadedMaterials : ARRAY[Surface.TOP..Surface.BOTTOM] OF STRING;
END_VAR
VAR CONSTANT
	sectionID : SectionEnum := SectionEnum.WOOD_BUNK;
END_VAR
VAR
	templateLeft, templateRight : AOI_StagingTemplate;
	stageLeft, stageRight : AOI_StageWoodBunk; 
	loadLeft, loadRight : AOI_LoadWoodBunk;
	
	topSuctionDelay : TON;
	
	a,b,c,d : BOOL;
	x : BOOL;
END_VAR

callLocalModules(); //initialize local modules

blocks(); //call local function blocks

IF robotRight.Done THEN
	robotRight.clearCommand();
END_IF

IF stop THEN
	stopSequence(); //stop everything
	RETURN;
END_IF
(*
IF NOT insertionLeft.screw.HomeSet OR NOT insertionRight.screw.HomeSet THEN
	homingSequence(); //homing all motion devices and robots
	RETURN;
END_IF
*)
a S= suctionTop[1].occupied AND suctionTop[2].occupied AND suctionTop[3].occupied;
b S= suctionLeft[1].occupied AND suctionLeft[2].occupied AND suctionLeft[3].occupied AND suctionLeft[4].occupied;
c S= suctionRight[1].occupied AND suctionRight[2].occupied AND suctionRight[3].occupied AND suctionRight[4].occupied;
d S= suctionBottom[1].occupied AND suctionBottom[2].occupied;

CASE step OF
	IDLE:
		IF execute THEN
			execute := FALSE;
			suctionEnableTop := suctionEnableLeft := suctionEnableRight := suctionEnableBottom := FALSE;
			step := STAGING;
		END_IF
		
		SetSuctions(suctionTop, suctionEnableTop);
		SetSuctions(suctionLeft, suctionEnableLeft);
		SetSuctions(suctionRight, suctionEnableRight);
		SetSuctions(suctionBottom, suctionEnableBottom);
		
	STAGING:
		IF NOT done THEN
			done := stage(); //calls stageEx() for both robots
		END_IF
		
		IF
			(manualStep AND_THEN execute) OR
			(NOT manualStep AND_THEN done)
		THEN
			robotLeft.clearCommand();
			robotRight.clearCommand();
			
			stageLeft.reset();
			stageRight.reset();
			
			execute := FALSE;
			done := FALSE;
			step := LOAD_WB;
		END_IF
	
	LOAD_WB:
		IF NOT done THEN
			done := load(pairIndex := iPair, error => error);
		END_IF
		
		IF manualSuction THEN
			SetSuctions(suctionTop, suctionEnableTop);
			SetSuctions(suctionLeft, suctionEnableLeft);
			SetSuctions(suctionRight, suctionEnableRight);
			SetSuctions(suctionBottom, suctionEnableBottom);
		END_IF
		
		IF
			(manualStep AND_THEN execute) OR
			(NOT manualStep AND_THEN done)
		THEN
			robotLeft.clearCommand();
			robotRight.clearCommand();
			
			done := FALSE;
			suctionEnableTop := suctionEnableLeft := suctionEnableRight := suctionEnableBottom := FALSE;
			execute := FALSE;
			
			step := PUSH;
		END_IF
		
	PUSH:
		IF
			(manualStep AND_THEN execute) OR
			(latchLeft AND latchRight AND pistonBottom.extended)
		THEN
			latchLeft := latchRight := FALSE;
			execute := FALSE;
			step := STRAP;
			RETURN;
		END_IF
		
		IF NOT validateSuctionQuality(checkTop:= TRUE, checkLeft:= TRUE, checkRight:= FALSE, checkBottom:= FALSE) THEN
			error := TRUE;
			RETURN;
		END_IF
		(*
		IF 
			insertionLeft.sliderPos <> demoHeight/2 //OR 
			//insertionRight.sliderPos <> demoHeight/2 //OR 
			//NOT insertionBottom.contact
		THEN
			insertionLeft.slideAbsolute(demoHeight/2);
			//insertionRight.slideAbsolute(demoHeight/2);
			RETURN;
		END_IF
		*)
		
		IF insertionLeft.screw.AtInnerLimit THEN
			latchLeft := TRUE;
		ELSIF NOT latchLeft THEN
			insertionLeft.press();
		END_IF
		
		IF insertionRight.screw.AtInnerLimit THEN
			latchRight := TRUE;
		ELSIF NOT latchRight THEN
			insertionRight.press();
		END_IF
		pistonBottom.extend();
		
	STRAP:
		topSuctionDelay(IN:= , PT:= T#1S, Q=> , ET=> );
		
		strapper.bEnable := TRUE;
		IF strapper.done THEN
			topSuctionDelay.IN := FALSE;
			step := RELEASE;
			RETURN;
		END_IF
		
		IF topSuctionDelay.Q THEN
			SetSuctions(suctionTop, FALSE);
			SetSuctions(suctionLeft, FALSE);
			SetSuctions(suctionRight, FALSE);
			SetSuctions(suctionBottom, FALSE);
		ELSIF strapper.atBundleLevel THEN
			topSuctionDelay.IN := TRUE;
		END_IF
		
		IF strapper.ready THEN
			strapper.strap();
		END_IF
		
		IF execute THEN
			topSuctionDelay.IN := FALSE;
			execute := FALSE;
			step := RELEASE;
		END_IF
		
	RELEASE: //release command		
		//insertionLeft.slideAbsolute(0);
		//insertionRight.slideAbsolute(0);
		
		insertionLeft.release();
		insertionRight.release();
		pistonBottom.retract();
		
		IF 
			(insertionLeft.screw.AtHome AND insertionRight.screw.AtHome AND pistonBottom.retracted) OR
			execute
		THEN
			execute := FALSE;
			step := COMPLETE;
		END_IF
	
	COMPLETE:
		//reset everything
		iPair := (iPair + 1) MOD GVL.maxPairs;
		step := IDLE;
		
		a := b := c := d := FALSE;
END_CASE

ACTION blocks:
templateLeft(
	execute:= , 
	materialsArr:= materialsArr, 
	table:= stagingTableLeft, 
	includeTop:= , 
	includeLeft:= , 
	includeRight:= , 
	includeBottom:= );

templateRight(
	execute:= , 
	materialsArr:= materialsArr, 
	table:= stagingTableRight, 
	includeTop:= , 
	includeLeft:= , 
	includeRight:= , 
	includeBottom:= );
	
stageLeft(
	sectionID:= sectionID, 
	execute:= ,
	robot:= robotLeft, 
	table:= stagingTableLeft, 
	magazine:= magazineLeft, 
	slot:= (*iSlotLeft*), 
	material:= templateLeft.getSlot(stageLeft.slot), 
	done=> , 
	error=> );

stageRight(
	sectionID:= sectionID, 
	execute:= ,
	robot:= robotRight, 
	table:= stagingTableRight, 
	magazine:= magazineRight, 
	slot:= (*iSlotRight*), 
	material:= templateRight.getSlot(stageRight.slot),
	done=> , 
	error=> );

loadLeft(
	sectionID:= sectionID, 
	execute:= ,
	robot:= robotLeft, 
	table:= stagingTableLeft, 
	suctions:= ,
	loadedMaterials:= loadedMaterials,
	//recoveryAoiStage:= stageLeft, 
	//recoveryMagazine:= magazineLeft, 
	surfaceID:= , 
	material:= , 
	loadedMaterials=> , 
	done=> , 
	error=> );
	
loadRight(
	sectionID:= sectionID, 
	execute:= ,
	robot:= robotRight, 
	table:= stagingTableRight, 
	suctions:= ,
	loadedMaterials:= loadedMaterials,
	//recoveryAoiStage:= stageRight, 
	//recoveryMagazine:= magazineRight, 
	surfaceID:= , 
	material:= , 
	loadedMaterials=> , 
	done=> , 
	error=> );
END_ACTION

ACTION callLocalModules:
{warning disable C0371}

insertionLeft(
	enable:= TRUE, 
	slider:= verticalDriveLeft, 
	screw:= horizontalDriveLeft, 
	contact=> , 
	softContact=> , 
	busy=> , 
	error=> , 
	home=> , 
	homingComplete=> , 
	sliderPos=> );
	
insertionRight(
	enable:= TRUE, 
	slider:= verticalDriveRight, 
	screw:= horizontalDriveRight,  
	contact=> , 
	softContact=> , 
	busy=> , 
	error=> , 
	home=> , 
	homingComplete=> , 
	sliderPos=> );
END_ACTION

ACTION homingSequence:
insertionLeft.homingSequence();
insertionRight.homingSequence();
pistonBottom.retract();
END_ACTION

METHOD PRIVATE load : BOOL
VAR_INPUT
	pairIndex : INT;
END_VAR
VAR_OUTPUT
	error : BOOL;
END_VAR
VAR
	pair : REFERENCE TO PositionMaterials REF= materialsArr[pairIndex];
END_VAR
{warning disable C0371}
IF robotLeft.error OR robotRight.error THEN
	error := TRUE;
	RETURN;
	
ELSIF 
	(robotLeft.reservation <> sectionID AND_THEN NOT robotLeft.reserve(sectionID)) OR 
	(robotRight.reservation <> sectionID AND_THEN NOT robotRight.reserve(sectionID))
THEN //loading requires both robots be reserved together
	RETURN;
	
ELSIF //robots have wrong tool
	(robotLeft.tool <> sectionID AND_THEN NOT robotLeft.changeEOAT(targetTool := sectionID)) OR
	(robotRight.tool <> sectionID AND_THEN NOT robotRight.changeEOAT(targetTool := sectionID))
THEN
	RETURN;
	
END_IF

CASE loadStep OF
	0: //top and bottom
		IF loadLeft.done AND loadRight.done THEN
			loadLeft.execute := loadRight.execute := FALSE;
			loadLeft.material := loadRight.material := '';
			loadStep := 10;
			RETURN;
		END_IF
		
		loadLeft.suctions := suctionTop;
		loadLeft.surfaceID := Surface.TOP;
		loadLeft.material := pair.top;
		
		loadRight.suctions := suctionBottom;
		loadRight.surfaceID := Surface.BOTTOM;
		loadRight.material := pair.bottom;
		
		loadLeft.execute := NOT loadLeft.done;
		loadRight.execute := NOT loadLeft.done;
		
	10: //sides
		IF
			(loadLeft.material = pair.left AND loadLeft.done) AND
			(loadRight.material = pair.right AND loadRight.done)
		THEN
			loadLeft.execute := loadRight.execute := FALSE;
			loadLeft.material := loadRight.material := '';
			loadStep := COMPLETE;
			RETURN;
		END_IF
		
		loadLeft.suctions := suctionLeft;
		loadLeft.surfaceID := Surface.LEFT;
		loadLeft.material := pair.left;
		
		loadRight.suctions := suctionRight;
		loadRight.surfaceID := Surface.RIGHT;
		loadRight.material := pair.right;
		
		loadLeft.execute := TRUE;
		loadRight.execute := TRUE;
		
	COMPLETE:				
		robotLeft.release(sectionID);
		robotRight.release(sectionID);
		
		loadLeft.material := loadRight.material := '';
		loadLeft.execute := loadRight.execute := FALSE;
		
		loadStep := 0;
		load := TRUE;
END_CASE

//--------------------------------------------------
IF loadLeft.recovery THEN //if loading in recovery mode - refill table, resume loading when finished
	loadLeft.execute := stageEx(
		robot:= robotLeft, 
		aoiTemplate:= templateLeft, 
		aoiStaging:= stageLeft, 
		stageStep:= stageStepLeft, 
		//iSlot:= iSlotLeft, 
		includeTop:= TRUE, 
		includeLeft:= TRUE, 
		includeRight:= FALSE, 
		includeBottom:= FALSE, 
		error=> );
ELSE
	//loadLeft.execute := NOT loadLeft.busy AND NOT loadLeft.done;
END_IF
//--------------------------------------------------
IF loadRight.recovery THEN
	loadRight.execute := stageEx(
		robot:= robotRight, 
		aoiTemplate:= templateRight, 
		aoiStaging:= stageRight, 
		stageStep:= stageStepRight, 
		//iSlot:= iSlotRight, 
		includeTop:= FALSE, 
		includeLeft:= FALSE, 
		includeRight:= TRUE, 
		includeBottom:= TRUE, 
		error=> );
ELSE
	//loadRight.execute := NOT loadRight.busy AND NOT loadRight.done;
END_IF
//--------------------------------------------------
	
error := loadLeft.error OR loadRight.error;
END_METHOD

METHOD PRIVATE stage : BOOL
VAR_OUTPUT
	error : BOOL;
END_VAR
{warning disable C0371}

(*
this method only exists to call stageEx() for both robots
*)

stage :=
	stageEx(
		robot:= robotLeft, 
		aoiTemplate:= templateLeft, 
		aoiStaging:= stageLeft, 
		stageStep:= stageStepLeft, 
		//iSlot:= iSlotLeft, 
		includeTop:= TRUE, 
		includeLeft:= TRUE, 
		includeRight:= FALSE, 
		includeBottom:= FALSE, 
		error=> )
	AND
	stageEx(
		robot:= robotRight, 
		aoiTemplate:= templateRight, 
		aoiStaging:= stageRight, 
		stageStep:= stageStepRight, 
		//iSlot:= iSlotRight, 
		includeTop:= FALSE, 
		includeLeft:= FALSE, 
		includeRight:= TRUE, 
		includeBottom:= TRUE, 
		error=> );
END_METHOD

METHOD PRIVATE stageEx : BOOL
VAR_IN_OUT
	robot : RobotA21;
	aoiTemplate : AOI_StagingTemplate;
	aoiStaging : AOI_StageWoodBunk;
	stageStep : INT;
	//iSlot : INT;
END_VAR
VAR_INPUT
	includeTop, includeLeft, includeRight, includeBottom : BOOL; 
END_VAR
VAR_OUTPUT
	error : BOOL;
END_VAR
{warning disable C0371}

IF robot.error THEN
	error := TRUE;
	RETURN;
ELSIF robot.reservation <> sectionID AND_THEN NOT robot.reserve(sectionID) THEN
	RETURN;
ELSIF robot.tool <> sectionID AND_THEN NOT robot.changeEOAT(targetTool := sectionID) THEN
	RETURN;
END_IF

CASE stageStep OF
	0: //generate staging template
		IF aoiTemplate.done THEN
			aoiTemplate.execute := FALSE;
			stageStep := 10;
			RETURN;
		END_IF
		
		aoiTemplate.execute := NOT aoiTemplate.busy;
		
		aoiTemplate.includeTop := includeTop;
		aoiTemplate.includeLeft := includeLeft;
		aoiTemplate.includeRight := includeRight;
		aoiTemplate.includeBottom := includeBottom;
		
	10: //stage tables
		IF aoiStaging.slot > 10 THEN
			aoiStaging.execute := FALSE;			
			stageStep := COMPLETE;
			RETURN;
		END_IF
		
		aoiStaging.slot := MAX(1, aoiStaging.slot); //if 0, sets to 1
		aoiStaging.slot := MIN(aoiStaging.slot, 999); //prevents overflow 
		
		aoiStaging.execute := NOT aoiStaging.busy; //execute if aoiStaging is ready
		
		IF aoiStaging.done THEN
			aoiStaging.slot := aoiStaging.slot + 1;
		END_IF
	
	COMPLETE:
		aoiTemplate.clearTemplate();
		aoiTemplate.execute := FALSE;
		aoiStaging.execute := FALSE;
		aoiStaging.reset();
		
		robot.release(sectionID);
		
		aoiStaging.slot := 0;
		
		stageEx := TRUE;
		//stageStep := 0;
END_CASE

error := aoiStaging.error;
END_METHOD

ACTION stopSequence:
insertionLeft.stop();
insertionRight.stop();
pistonBottom.stop();

robotLeft.clearCommand();
robotRight.clearCommand();

//stop conveyors
END_ACTION

METHOD PRIVATE validateSuctionQuality : BOOL
VAR_INPUT
	checkTop : BOOL;
	checkLeft : BOOL;
	checkRight : BOOL;
	checkBottom : BOOL;
END_VAR
validateSuctionQuality := 
	(NOT checkTop OR_ELSE SuctionQuality(suctions:= suctionTop)) AND
	(NOT checkLeft OR_ELSE SuctionQuality(suctions:= suctionLeft)) AND
	(NOT checkRight OR_ELSE SuctionQuality(suctions:= suctionRight)) AND
	(NOT checkBottom OR_ELSE SuctionQuality(suctions:= suctionBottom));

(*
validateSuctionQuality := 
	(
		NOT checkTop OR_ELSE InsertionQuality(
			suctions:= suctionTop, 
			insertionMaterial:= loadedMaterials[Surface.TOP], 
			recipeMaterial:= materialsArr[iPair].top)
	) AND
	(
		NOT checkLeft OR_ELSE InsertionQuality(
			suctions:= suctionLeft, 
			insertionMaterial:= loadedMaterials[Surface.LEFT], 
			recipeMaterial:= materialsArr[iPair].left)
	) AND
	(
		NOT checkRight OR_ELSE InsertionQuality(
			suctions:= suctionRight, 
			insertionMaterial:= loadedMaterials[Surface.RIGHT], 
			recipeMaterial:= materialsArr[iPair].right)
	) AND
	(
		NOT checkBottom OR_ELSE InsertionQuality(
			suctions:= suctionBottom, 
			insertionMaterial:= loadedMaterials[Surface.BOTTOM], 
			recipeMaterial:= materialsArr[iPair].bottom)
	);
*)
END_METHOD

END_FUNCTION_BLOCK

// ---- POUs/A21b - Wood Bunk/AOIs/AOI_StagingTemplate.TcPOU
FUNCTION_BLOCK AOI_StagingTemplate
VAR_INPUT
	execute : BOOL;
END_VAR
VAR_IN_OUT
	materialsArr : ARRAY[*] OF PositionMaterials; //[0..GVL.maxPairs]
	table : StagingTable;
END_VAR
VAR_INPUT
	includeTop, includeLeft, includeRight, includeBottom : BOOL; 
END_VAR
VAR_OUTPUT
	busy : BOOL;
	done : BOOL;
END_VAR
VAR
	trigger : R_TRIG;
	run : BOOL;
	step : (IDLE, GENERATE, COMPLETE);
	i : INT;
END_VAR
VAR	
	stagingArray : ARRAY[0..(GVL.maxPairs+1)*2] OF STRING;
	template : StagingTable;
	templateSlots : ARRAY[1..10] OF STRING;
	templateOccupancy : ARRAY[1..10] OF BOOL;
END_VAR

{warning disable C0371}

template(slots:= templateSlots, occupied:= templateOccupancy);

trigger(CLK:= execute, Q=> run);

CASE step OF
	IDLE:
		IF run THEN
			step := GENERATE;
			done := FALSE;
		END_IF
		
	GENERATE:
		//if staging array is empty, then fill the array
		//strings contain garbage chars after a null byte, they must be manually cleaned before checking if they are byte-empty
		CleanStringsArray(arr := stagingArray);
		IF ArrayIsEmpty(arr := ADR(stagingArray), arrSize := SIZEOF(stagingArray)) THEN
			createStagingArray(
				includeTop:= includeTop, 
				includeLeft:= includeLeft, 
				includeRight:= includeRight, 
				includeBottom:= includeBottom);
		END_IF
		
		//copy over the real slots before autofilling, otherwise the template may fill occupied slots
		MEMCPY(template.slots, table.slots, SIZEOF(STRING) * 10);
		
		(*
		iterate through all pairs and autofill the template
		replace succesfully autofilled materials with empty string
		if staging needs to be performed a 2nd time, autofilling empty strings is always unsuccessful
		*)
		FOR i:=0 TO (GVL.maxPairs+1)*2 BY 1 DO
			IF template.autofill(materialID := stagingArray[i]) THEN
				stagingArray[i] := '';
			END_IF
		END_FOR
		
		step := COMPLETE;
	
	COMPLETE:
		done := TRUE;
		
		step := IDLE;
		
END_CASE

busy := run OR step > 0;

METHOD PRIVATE addToStagingArray : BOOL
VAR_INPUT
	material : STRING;
END_VAR
VAR
	remainingMaterial : STRING;
	splitMaterial : STRING;
END_VAR
remainingMaterial := material;
WHILE FIND(remainingMaterial, '_') > 0 DO
	splitCombinedMaterials(remainingMaterial, splitMaterial);
	IF splitMaterial <> '' THEN
		AddToStringArray(arr := stagingArray, newString := splitMaterial, numElements => , nextIndex => );
	END_IF
END_WHILE

IF remainingMaterial <> '' THEN
	AddToStringArray(arr := stagingArray, newString := remainingMaterial, numElements => , nextIndex => );
END_IF

addToStagingArray := TRUE;
END_METHOD

METHOD clearArray : BOOL
VAR_INPUT
END_VAR
MEMSET(ADR(stagingArray), 0, SIZEOF(stagingArray));
END_METHOD

METHOD clearTemplate : BOOL
VAR_INPUT
END_VAR
template.clear();
END_METHOD

METHOD PRIVATE createStagingArray : BOOL
VAR_INPUT
	includeTop : BOOL;
	includeLeft : BOOL;
	includeRight : BOOL;
	includeBottom : BOOL;
END_VAR
VAR
	remainingMaterial : STRING;
	splitMaterial : STRING;
	
	i : INT;
END_VAR
FOR i:=0 TO GVL.maxPairs BY 1 DO
	IF includeTop THEN
		addToStagingArray(material := materialsArr[i].top);
	END_IF
	
	IF includeLeft THEN
		addToStagingArray(material := materialsArr[i].left);
	END_IF
	
	IF includeRight THEN
		addToStagingArray(material := materialsArr[i].right);
	END_IF
	
	IF includeBottom THEN
		addToStagingArray(material := materialsArr[i].bottom);
	END_IF
END_FOR
END_METHOD

METHOD getSlot : STRING
VAR_INPUT
	i : INT;
END_VAR
VAR_OUTPUT
	error : BOOL;
END_VAR
getSlot := template.getSlot(i := i, error => error);
END_METHOD

METHOD reset : BOOL
VAR_INPUT
END_VAR
VAR
	temp : AOI_StagingTemplate;
END_VAR
//(*
busy := FALSE;
done := FALSE;
step := 0;

clearArray();
clearTemplate();
//*)
//THIS^ := temp;
END_METHOD

METHOD PRIVATE splitCombinedMaterials : BOOL
VAR_IN_OUT
	materialID : STRING;
	splitMaterial : STRING;
END_VAR
VAR
	i : INT;
END_VAR
FindAndSplitChar(
	sSeparatorChar:= '_', 
	pSrcString:= ADR(materialID), 
	
	pLeftString:= ADR(splitMaterial), 
	nLeftSize:= SIZEOF(splitMaterial), 
	
	pRightString:= ADR(materialID), 
	nRightSize:= SIZEOF(materialID), 
	
	bSearchFromRight:= FALSE);
END_METHOD

END_FUNCTION_BLOCK

// ---- POUs/A21b - Wood Bunk/AOIs/AOI_StageWoodBunk.TcPOU
FUNCTION_BLOCK AOI_StageWoodBunk
VAR_IN_OUT CONSTANT
	sectionID : SectionEnum;
END_VAR
VAR_INPUT
	execute : BOOL;
END_VAR
VAR_IN_OUT
	robot : RobotA21;
	table : StagingTable;
	magazine : SkidMagazine;
END_VAR
VAR_INPUT
	slot : INT;
	material : STRING;
END_VAR
VAR_OUTPUT
	busy : BOOL;
	done : BOOL;
	error : BOOL;
	
	recovery : BOOL;
	failCounter : INT;
END_VAR
VAR
	trigger : R_TRIG;
	run : BOOL;
	
	magazineColumn : INT;
	step : (IDLE, PREP_ROBOT, GET_FROM_MAGAZINE, PLACE_ON_TABLE, COMPLETE);
END_VAR
VAR CONSTANT
	suctionDistance : INT := 10;
END_VAR

{warning disable C0371}
{warning disable C0195}

//--------------------------------------------------

trigger(CLK:= execute, Q=> );
busy := trigger.Q OR step > 0;

IF step > IDLE AND_THEN NOT preExecution() THEN //conditions to track before execution
	RETURN;
END_IF

//follow the template as is
CASE step OF
	IDLE:
		recovery := FALSE;
		IF trigger.Q THEN
			done := FALSE;
			error := FALSE;
			step := PREP_ROBOT;
		END_IF
		
	PREP_ROBOT:
		robot.clearCommand();
		IF robot.Ready THEN
			step := GET_FROM_MAGAZINE;
		END_IF
	
	GET_FROM_MAGAZINE: //grab from magazine
		IF NOT magazine.findSlot(materialID := material, index => magazineColumn) THEN
			error := TRUE;
			RETURN;
		END_IF
		
		IF robot.eoatDistance < suctionDistance THEN //robot is grabbing material
			robot.HoldMaterial := magazine.getSlot(i := magazineColumn);
		END_IF
		
		IF robot.Done THEN
			step := COMPLETE;
			RETURN;
		END_IF
		
		robot.setGroup(group := 1, value := A21.STAGE_BUNK);
		robot.setGroup(group := 2, value := magazineColumn);
		robot.setGroup(group := 3, value := slot);

	COMPLETE: //check here if staging is successful or needs to be repeated
		robot.clearCommand();
		
		IF table.isOccupied(slot) THEN
			table.place(i := slot, materialID := robot.HoldMaterial);
			robot.HoldMaterial := '';
			
			failCounter := 0;
			done := TRUE;
		ELSE
			failCounter := failCounter + 1;
		END_IF
		
		step := 0;
		
END_CASE

METHOD PRIVATE preExecution : BOOL
VAR_INPUT
END_VAR
{warning disable C0371}

IF slot < 1 THEN //out of bounds for staging table
	error := TRUE;
	RETURN;
ELSIF table.isFull() OR slot > 10 OR material = '' OR table.getSlot(i := slot, error => ) = material THEN
	done := TRUE;
	RETURN;
END_IF

IF //robot must be ready before execution
	robot.error OR 
	robot.reservation <> sectionID OR 
	robot.tool <> sectionID
THEN
	error := TRUE;
	RETURN;
END_IF

preExecution := TRUE;
END_METHOD

METHOD reset : BOOL
VAR_INPUT
END_VAR
done := FALSE;
error := FALSE;
slot := 0;
step := 0;

failCounter := 0;
END_METHOD

END_FUNCTION_BLOCK

// ---- POUs/A21a - Chipboard/ChipboardEx.TcPOU
FUNCTION_BLOCK ChipboardEx
VAR_IN_OUT //controls
	execute : BOOL;
	stop : BOOL;
	
	manualStep : BOOL;
END_VAR
VAR_IN_OUT //references to required hardware
	robotLeft, robotRight : RobotA21;
	toolStorageLeft, toolStorageRight : A21ToolStorage;
	
	skidLeft, skidRight : SkidMagazine;
END_VAR
VAR_OUTPUT
	//ready : BOOL;
	done : BOOL;
	generalError : BOOL;
	failLeft, failRight : BOOL;
END_VAR
VAR //for testing, to be removed when replaced with pressure sensors
	latchLeft, latchRight : BOOL;
	
	demoHeight : REAL := 600; //mm
END_VAR
VAR
	step : (IDLE, RETRACT_CONVEYOR, LOAD_CIP, EXTEND_CONVEYOR, COMPLETE := 1050);
	iPair : INT;
	
	loadSet : INT;
END_VAR
VAR //local types
	materialsArr : ARRAY[0..GVL.maxPairs] OF PositionMaterials := [
		(position := 0, top := 'CIP54', bottom := 'CIP18')
	];
		
	loadedMaterials : ARRAY[Surface.TOP..Surface.BOTTOM] OF STRING;
END_VAR
VAR CONSTANT
	sectionID : SectionEnum := SectionEnum.CHIPBOARD;
END_VAR
VAR
	loadLeft, loadRight : AOI_LoadChipboard;
END_VAR

{warning disable C0371}
callLocalModules();

IF stop THEN //may need to turn off suction	
	robotLeft.clearCommand();
	robotRight.clearCommand();
	RETURN;
END_IF

IF FALSE (*conveyors not extended*) THEN
	RETURN;
END_IF

CASE step OF
	IDLE:
		IF execute THEN
			execute := FALSE;
			step := RETRACT_CONVEYOR;
		END_IF
		
	RETRACT_CONVEYOR:
		(*
		IF demoPair.bottom <> '' (*retract conveyors*) THEN
			IF TRUE (*BLSC 1-3 retracted*) THEN
				done := TRUE;
			END_IF
		ELSE
			done := TRUE;
		END_IF
		
		IF
			(manualStep AND_THEN execute) OR
			(NOT manualStep AND_THEN done)
		THEN
			done := FALSE;
			step := LOAD_MATERIAL;
		END_IF
		*)
		step := LOAD_CIP;
	LOAD_CIP:
		IF NOT done THEN
			done := load(pairIndex:= iPair, error=> generalError);
		END_IF
		
		IF
			(manualStep AND_THEN execute) OR
			(NOT manualStep AND_THEN done)
		THEN
			done := FALSE;
			execute := FALSE;
			
			step := EXTEND_CONVEYOR;
		END_IF
		
	EXTEND_CONVEYOR:
		(*
		IF FALSE (*conveyors not extended*) THEN
			//extend conveyors
		END_IF
		
		IF
			(manualStep AND_THEN execute) OR
			(FALSE) //conveyors extended
		THEN
			done := FALSE;
			step := COMPLETE;
		END_IF
		*)
		step := COMPLETE;
	COMPLETE:
		//reset everything
		step := IDLE;
		
END_CASE

ACTION blocks:
loadRight(
	sectionID:= sectionID, 
	execute:= ,
	robot:= robotRight, 
	storage:= skidRight,
	loadedMaterials:= loadedMaterials,
	surfaceID:= , 
	material:= , 
	loadedMaterials=> , 
	done=> , 
	error=> );
	
loadRight(
	sectionID:= sectionID, 
	execute:= , 
	robot:= robotRight, 
	storage:= skidRight,
	loadedMaterials:= loadedMaterials, 
	surfaceID:= , 
	material:= , 
	busy=> , 
	done=> , 
	error=> , 
	recovery=> , 
	failCounter=> );
END_ACTION

METHOD PRIVATE callLocalModules : BOOL
END_METHOD

METHOD PRIVATE load : BOOL
VAR_INPUT
	pairIndex : INT;
END_VAR
VAR_OUTPUT
	error : BOOL;
END_VAR
VAR
	pair : REFERENCE TO PositionMaterials REF= materialsArr[pairIndex];
END_VAR
{warning disable C0371}
IF robotLeft.error AND robotLeft.error THEN
	error := TRUE;
	RETURN;

ELSIF
	( robotLeft.reservation <> sectionID AND_THEN robotLeft.reserve(sectionID) ) OR
	( robotRight.reservation <> sectionID AND_THEN robotRight.reserve(sectionID) ) THEN
	RETURN;
	
ELSIF //wrong tool and not finished changing tool
	(robotLeft.tool <> sectionID AND_THEN NOT robotLeft.changeEOAT(targetTool := sectionID)) OR
	(robotRight.tool <> sectionID AND_THEN NOT robotRight.changeEOAT(targetTool := sectionID))
THEN
	RETURN;
END_IF
//robots ok

CASE loadSet OF
	0: //left robot -> top, right robot -> bottom
		IF loadLeft.done AND loadRight.done THEN
			loadLeft.execute := loadRight.execute := FALSE;
			loadSet := 10;
			RETURN;
		END_IF
		
		loadLeft.surfaceID := Surface.TOP;
		loadLeft.material := pair.left;
		
		loadRight.surfaceID := Surface.BOTTOM;
		loadRight.material := pair.right;
		
		loadLeft.execute := NOT loadLeft.recovery;
		loadRight.execute := NOT loadRight.recovery;
		
	10: //recovery		
		IF robotRight.error THEN //left ok, right error
			
			IF loadLeft.done THEN
				loadLeft.execute := FALSE;
				loadSet := COMPLETE;
				RETURN;
			END_IF
			
			loadLeft.surfaceID := Surface.BOTTOM;
			loadLeft.material := pair.bottom;
			loadLeft.execute := NOT loadLeft.recovery;
			
		ELSIF robotLeft.error THEN //left error, right ok
			
			IF loadRight.done THEN
				loadRight.execute := FALSE;
				loadSet := COMPLETE;
				RETURN;
			END_IF
			
			loadRight.surfaceID := Surface.TOP;
			loadRight.material := pair.top;
			loadRight.execute := NOT loadRight.recovery;
			
		END_IF
		
	COMPLETE:
		loadSet := 0;
		
		robotLeft.release(sectionID);
		robotRight.release(sectionID);
		
		load := TRUE;
END_CASE
END_METHOD

METHOD PRIVATE loadingSequence : BOOL
VAR_IN_OUT
	robot : RobotA21;
	storage : SkidMagazine;
	loadStep : INT;
END_VAR
VAR_INPUT
	surfaceID : Surface;
	material : STRING;
END_VAR
VAR_OUTPUT
	fail : BOOL;
END_VAR
VAR
	slot : INT;
END_VAR
VAR CONSTANT
	suctionDistance : INT := 10;
END_VAR
{warning disable C0371}
IF material = '' THEN
	loadingSequence := TRUE;
	RETURN;
END_IF

CASE loadStep OF
	0:
		robot.clearCommand();
		IF robot.Ready THEN
			loadStep := 1;
		END_IF
	
	1:
		IF surfaceID = Surface.BOTTOM (*AND_THEN conveyors not retracted*) THEN
			//retract conveyors
			RETURN;
		END_IF
		loadStep := 10;
		
	10: //grab from chipboard skid
		IF NOT storage.findSlot(materialID := material, index => slot) THEN
			fail := TRUE;
			RETURN;
		(*
		ELSIF surfaceID = Surface.BOTTOM (*AND_THEN (*conveyor not lowered*)*) THEN
			//lower conveyor
			RETURN;
		*)
		END_IF
		
		IF robot.eoatDistance < suctionDistance THEN
			robot.HoldMaterial := storage.getSlot(i := slot);
		END_IF
		
		IF robot.Done THEN
			loadStep := COMPLETE;
			RETURN;
		ELSIF robot.materialAtHoldingPosition.4 OR robot.materialAtHoldingPosition.5 THEN //bits 4 and 5 are chipboard in position
			loadStep := 20;
			RETURN;
		END_IF
		
		robot.setGroup(group := 1, value := A21.PLACE_CHIPBOARD_TOP);
		robot.setGroup(group := 2, value := slot);
		
	20: //place to bundle
		IF robotLeft.Done THEN
			loadStep := COMPLETE;
			RETURN;
		END_IF
		
		IF robot.HoldMaterial <> '' THEN
			loadedMaterials[surfaceID] := robot.HoldMaterial;
			robot.HoldMaterial := '';
		END_IF
		
	COMPLETE:
		IF loadedMaterials[surfaceID] = material THEN
			loadingSequence := TRUE;
		ELSE
			loadStep := 0;
		END_IF
		
END_CASE
END_METHOD

END_FUNCTION_BLOCK

// ---- POUs/Hardware Calls/CallHardware.TcPOU
FUNCTION CallHardware : BOOL //only purpose of this function is to call modules from Hardware
VAR_STAT
	tempLeft, tempRight : INT;
END_VAR

robot1();	
robot2();

skidA21Left(slots := skidSlotsA21Left, occupied := skidOccupancyA21Left, hmiTable := skidHmiA21Left);
skidA21Right(slots := skidSlotsA21Right, occupied := skidOccupancyA21Right, hmiTable := skidHmiA21Right);

stagingTableLeft(slots := tableSlotsA21Left, occupied := tableOccupancyA21Left, hmiTable := tableHmiA21Left);
stagingTableRight(slots := tableSlotsA21Right, occupied := tableOccupancyA21Right, hmiTable := tableHmiA21Right);

magazineA21Left(slots := magazineSlotsA21Left, occupied := magazineOccupancyA21Left, hmiTable := magazineHmiA21Left);
magazineA21Right(slots := magazineSlotsA21Right, occupied := magazineOccupancyA21Right, hmiTable := magazineHmiA21Right);

strapperA21();

verticalDriveA21Left();
verticalDriveA21Right();
horizontalDriveA21Left();
horizontalDriveA21Right();
pistonA21Bottom();

(*
tempLeft := TO_INT(BoolPtrArrayToInteger(arr := stagingTableLeft.occupied, lowerBound := 1, upperBound := 10));
tempLeft.15 := NOT strapperA21.bEnable AND NOT strapperA21.execute;
robot1.setGroup(group := 8, value := tempLeft);

tempRight := TO_INT(BoolPtrArrayToInteger(arr := stagingTableRight.occupied, lowerBound := 1, upperBound := 10));
tempRight.15 := NOT strapperA21.bEnable AND NOT strapperA21.execute;
robot2.setGroup(group := 8, value := tempRight);

*)

END_FUNCTION

// ---- POUs/Hardware Calls/SetupHardware.TcPOU
FUNCTION SetupHardware : BOOL
VAR
	iWoodBunkSlot : WoodBunk;
	iChipboardSlot : Chipboard;
	
	i : INT;
END_VAR

FOR iWoodBunkSlot:=1 TO WoodBunk.size-1 BY 1 DO //init wood bunk magazine slots
	magazineA21Left.setSlot(i := iWoodBunkSlot, material := TO_STRING(iWoodBunkSlot), error => );
	magazineA21Right.setSlot(i := iWoodBunkSlot, material := TO_STRING(iWoodBunkSlot), error => );
END_FOR

//--------------------------------------------------

FOR iChipboardSlot:=1 TO Chipboard.size-1 BY 1 DO //init chipboard skid slots
	skidA21Left.setSlot(i := iChipboardSlot, material := TO_STRING(iChipboardSlot), error => );
	skidA21Right.setSlot(i := iChipboardSlot, material := TO_STRING(iChipboardSlot), error => );
END_FOR

//--------------------------------------------------

FOR i:=1 TO GVL.maxQueue BY 1 DO //get wood bunk magazine + chipboard skid availability from robot1 and robot2
	{warning disable C0195}
	skidA21Left.setOccupancy( i := i, occupancy := IntegerBitAccess(robot1.inputs[4], i-1) );
	skidA21Right.setOccupancy( i := i, occupancy := IntegerBitAccess(robot2.inputs[4], i-1) );

	magazineA21Left.setOccupancy( i := i, occupancy := IntegerBitAccess(robot1.inputs[3], i-1) );
	magazineA21Right.setOccupancy( i := i, occupancy := IntegerBitAccess(robot2.inputs[3], i-1) );
END_FOR

//--------------------------------------------------

//enable all drives
verticalDriveA21Left.bEnable := 
verticalDriveA21Right.bEnable := 
horizontalDriveA21Left.bEnable := 
horizontalDriveA21Right.bEnable := 
pistonA21Bottom.bEnable := 
TRUE;

END_FUNCTION
